PROGRAM Hardware
VAR
	//Inputmodules:
	EL1004_X1 	AT%I*	: DIOmodule; //Käytetään tyyppinä struktuuria, joka on määritelty globaaleissa muuttujissa. Ks GVL
	EL1008_X2	AT%I*	: DIOmodule;
	
	//Outputmodules:
	EL2004_X3	AT%Q*	: DIOmodule;
	EL2008_X4	AT%Q*	: DIOmodule;
END_VAR

//Tulokanavien kytkeminen muuttujiin:
GVL.safetyOk 	:= EL1004_X1.input[0] ; //Tulokanava määrää muuttujan tilan
GVL.start		:= EL1008_X2.input[3] ;
GVL.stop		:= EL1008_X2.input[4] ;

//Muuttujien kytkeminen lähtökanaviin:
EL2004_X3.output[0] := GVL.stopBtnLight; //Muuttuja määrää lähtökanavan tilan
EL2004_X3.output[1] := GVL.startBtnLight;

END_PROGRAM

(* stored: Version 1.1.0.1, ProductVersion 3.1.4024.11
   POU Hardware: Id {5f71b22e-f98d-4df7-b852-44da5dd2b04a}, SpecialFunc None *)
